FUNCTION wordArray2DINT : DINT
VAR_INPUT
	wordLeft : WORD;
	wordRight : WORD; 
END_VAR
VAR
	wordArray : ARRAY [1..2] OF WORD;
	ptdint : POINTER TO DINT;
END_VAR

wordArray[2] := wordLeft;
wordArray[1] := wordRight;
ptdint := ADR(wordArray[1]);
wordArray2DINT := ptdint^;

END_FUNCTION

(* stored: Version 1.1.0.1, ProductVersion 3.1.0.36
   POU wordArray2DINT: Id {32b4643b-7960-4505-9459-810173506016}, SpecialFunc None *)
